// TIA Portal V16 export
// export: Created 2021-06-17T11:14:34.052257Z, ExportSetting WithDefaults, DisplayName Totally Integrated Automation Portal, DisplayVersion V16 Update 4, DisplayName TIA Portal Version Control Interface, DisplayVersion V16 Update 2, DisplayName TIA Portal Openness, DisplayVersion V16 Update 4, DisplayName SINAMICS Startdrive Advanced, DisplayVersion V16 Update 5, DisplayName SINAMICS Startdrive G130, G150, S120, S150, SINAMICS MV, S210, DisplayVersion V16 Update 5, DisplayName SINAMICS Startdrive G110M, G120, G120C, G120D, G120P, G115D, DisplayVersion V16 Update 5, DisplayName STEP 7 Professional, DisplayVersion V16 Update 4, DisplayName SIMATIC Energy Suite, DisplayVersion V16 Update 4, DisplayName STEP 7 Safety, DisplayVersion V16, DisplayName WinCC Advanced / Unified PC, DisplayVersion V16 Update 4, DisplayName SIMATIC Visualization Architect, DisplayVersion V16 Update 1
TYPE "UDT_ACB_ETI"
// stored: IsFailsafeCompliant false
   STRUCT
      ID : Int;   // MOT(ID=5001...6000)
      CLSID : Word := WORD#16#2110;   // Type of element
      Mode { ExternalAccessible := 'False'; ExternalVisible := 'False'; ExternalWritable := 'False'} : "Mode";
      State { ExternalAccessible := 'False'; ExternalVisible := 'False'; ExternalWritable := 'False'} : Struct   // Main state
         Error { ExternalAccessible := 'False'; ExternalVisible := 'False'; ExternalWritable := 'False'} : Bool;   // 1 = [1-level alarm] General alarm - Overall error
         Warning { ExternalAccessible := 'False'; ExternalVisible := 'False'; ExternalWritable := 'False'} : Bool;   // 1 = [2-level alarm] Warning
         Maintenance { ExternalAccessible := 'False'; ExternalVisible := 'False'; ExternalWritable := 'False'} : Bool;   // 1 = [3-level ] Maintenance
         Interlocked { ExternalAccessible := 'False'; ExternalVisible := 'False'; ExternalWritable := 'False'} : Bool;   // 1 = [Interlock] -Status interlock - Motor interlocked
         Ready { ExternalAccessible := 'False'; ExternalVisible := 'False'; ExternalWritable := 'False'} : Bool;   // 1 = Ready
         Closed { ExternalAccessible := 'False'; ExternalVisible := 'False'; ExternalWritable := 'False'} : Bool;   // 1 = Closed = IB_114_FeedbackClose+ QB_CmdCloseACB
         Opened { ExternalAccessible := 'False'; ExternalVisible := 'False'; ExternalWritable := 'False'} : Bool;   // 1 = Opened = IB_114_FeedbackOpen+ QB_CmdOpenACB
         Closing { ExternalAccessible := 'False'; ExternalVisible := 'False'; ExternalWritable := 'False'} : Bool;   // 1 = Closing - закривається
         Opening { ExternalAccessible := 'False'; ExternalVisible := 'False'; ExternalWritable := 'False'} : Bool;   // 1 = Opening - відкривається
         InCmdAutoClose { ExternalAccessible := 'False'; ExternalVisible := 'False'; ExternalWritable := 'False'} : Bool;   // 1 = Auto COMMAND - ACB to CLOSE
         InCmdAutoOpen { ExternalAccessible := 'False'; ExternalVisible := 'False'; ExternalWritable := 'False'} : Bool;   // 1 = Auto COMMAND - ACB to OPEN
         SigOutOpen { ExternalAccessible := 'False'; ExternalVisible := 'False'; ExternalWritable := 'False'} : Bool;   // StateTransferredTo physical output.Activate the output - QB_CmdCloseACB
         SigOutClose { ExternalAccessible := 'False'; ExternalVisible := 'False'; ExternalWritable := 'False'} : Bool;   // State transferred to physical output.Activate the output - QB_CmdOpenACB
      END_STRUCT;
      Alarm { ExternalAccessible := 'False'; ExternalVisible := 'False'; ExternalWritable := 'False'} : Struct
         InterlockingBypassed { ExternalAccessible := 'False'; ExternalVisible := 'False'; ExternalWritable := 'False'} : Bool;
         InterlockBypassed { ExternalAccessible := 'False'; ExternalVisible := 'False'; ExternalWritable := 'False'} : Bool;
         ErrTimeOut { ExternalAccessible := 'False'; ExternalVisible := 'False'; ExternalWritable := 'False'} : Bool;   // 1 = TimeOut
         ExtWarning { ExternalAccessible := 'False'; ExternalVisible := 'False'; ExternalWritable := 'False'} : Bool;   // 1 = External warning active + Warning
         ExtError { ExternalAccessible := 'False'; ExternalVisible := 'False'; ExternalWritable := 'False'} : Bool;   // 1 = External Fault is active + Error
         PreAlarm { ExternalAccessible := 'False'; ExternalVisible := 'False'; ExternalWritable := 'False'} : Bool;
         SystemFault { ExternalAccessible := 'False'; ExternalVisible := 'False'; ExternalWritable := 'False'} : Bool;   // 2^9 1 = Emergency SAFETY Motor Local switch OFF(Local disconnect OFF) +Error
         TripLT { ExternalAccessible := 'False'; ExternalVisible := 'False'; ExternalWritable := 'False'} : Bool;   // 2^10 0 = Motor Protector OK / 1 = Motor ProtectorTripped + Error
         TripST { ExternalAccessible := 'False'; ExternalVisible := 'False'; ExternalWritable := 'False'} : Bool;   // 2^11 0 = Clutch OK /1 = Clutch tripped + Error
         ErrClosing { ExternalAccessible := 'False'; ExternalVisible := 'False'; ExternalWritable := 'False'} : Bool;   // 2^12 1 = ÐŸÐ¾Ð¼Ð¸Ð»ÐºÐ° Ð·Ð°Ð¿ÑƒÑÐºÑƒ/ No signal from forward contactor + Error
         ErrOpening { ExternalAccessible := 'False'; ExternalVisible := 'False'; ExternalWritable := 'False'} : Bool;   // 2^141 = ÐŸÐ¾Ð¼Ð¸Ð»ÐºÐ° Ð·ÑƒÐ¿Ð¸Ð½ÐºÐ¸ / Motor doesn't stop / Switching time exceeded. + Error
         ErrPlaus { ExternalAccessible := 'False'; ExternalVisible := 'False'; ExternalWritable := 'False'} : Bool;   // 2^15 1=errorPlaus-Activation not plausible(switched on or switched off at the s
         MaintACT { ExternalAccessible := 'False'; ExternalVisible := 'False'; ExternalWritable := 'False'} : Bool;   // 2^6 1=Ðœaintenance-Limit Number object switching operations Reached + Maintenanc
         MaintTIME { ExternalAccessible := 'False'; ExternalVisible := 'False'; ExternalWritable := 'False'} : Bool;   // 2^7 1 = Ðœaintenance-Limit Operating time Reached + Maintenance
         EstopLocal { ExternalAccessible := 'False'; ExternalVisible := 'False'; ExternalWritable := 'False'} : Bool;   // 2^0 1 = Estop active + Error
         EstopHMI { ExternalAccessible := 'False'; ExternalVisible := 'False'; ExternalWritable := 'False'} : Bool;   // 2^0 1 = Estop active + Error
         FaultSuppyBox { ExternalAccessible := 'False'; ExternalVisible := 'False'; ExternalWritable := 'False'} : Bool;
      END_STRUCT;
      CMD : Int;   // 16#0100/16#0101/16#0102/16#0200/16#0201/16#0202/16#0300/16#0301/16#0302
      PRM : Struct
         W { ExternalAccessible := 'False'; ExternalVisible := 'False'; ExternalWritable := 'False'} : Struct
            ManLocalPirority { ExternalAccessible := 'False'; ExternalVisible := 'False'; ExternalWritable := 'False'; S7_SetPoint := 'True'} : Bool;   // 1 = HIGHT - enable from FC input/0 = LOW - enable from HMI
            AutoAskErrors { ExternalAccessible := 'False'; ExternalVisible := 'False'; ExternalWritable := 'False'; S7_SetPoint := 'True'} : Bool;   // 1 = Ð°Ð²Ñ‚Ð¾Ð¼Ð°Ñ‚Ð¸Ñ‡Ð½Ðµ Ð¿Ñ–Ð´Ñ‚Ð²ÐµÑ€Ð´Ð¶ÐµÐ½Ð½Ñ Ñ‚Ñ€Ð¸Ð²Ð¾Ð³
            LockExtModeChange { ExternalAccessible := 'False'; ExternalVisible := 'False'; ExternalWritable := 'False'; S7_SetPoint := 'True'} : Bool;
            InterlockBypass { ExternalAccessible := 'False'; ExternalVisible := 'False'; ExternalWritable := 'False'; S7_SetPoint := 'True'} : Bool;   // Interlocking obj bypassed / disable
            InterlockAutoReset { ExternalAccessible := 'False'; ExternalVisible := 'False'; ExternalWritable := 'False'; S7_SetPoint := 'True'} : Bool;
         END_STRUCT;
         enableExternalErrors { ExternalAccessible := 'False'; ExternalVisible := 'False'; ExternalWritable := 'False'; S7_SetPoint := 'True'} : Word := 16#FFFF;   // bit - 1 = enable
         bypassInterlocks { ExternalAccessible := 'False'; ExternalVisible := 'False'; ExternalWritable := 'False'; S7_SetPoint := 'True'} : Word := 16#FFFF;   // bit - 0 = Interlock Bypassed
         spTimeOut { S7_SetPoint := 'True'} : Int := 50;   // Monitoring time for ERROR ErrRunFRD ErrRunRVS ErrStop ErrPlaus (0.1sec)
         spTimeOnDelAuto { S7_SetPoint := 'True'} : Int := 50;   // Setpoint delay on time after start auto command (0.1sec)
         spTimeOffDelAuto { S7_SetPoint := 'True'} : Int := 50;   // Setpoint delay off time after stop auto command (0.1sec)
         spTimeRestart { S7_SetPoint := 'True'} : Int := 50;   // Час блокування повторного запуску (0.1sec)
         spTimeFixError { S7_SetPoint := 'True'} : Int := 50;   // Чac блокування скидання помилок дляїх фіксації в HMI (0.1sec.)
         spTimeCmdCloseOpen { S7_SetPoint := 'True'} : Int := 50;
         spMaintTimeOperPeriod { S7_SetPoint := 'True'} : DInt;   // Maintenance period - Operating time in hours 0=OFF (hour)
         spMaintActivPeriod { S7_SetPoint := 'True'} : DInt;   // Maintenance period-number object activated switches/switching operations 0=OFF
         spare48 { S7_SetPoint := 'True'} : Int;
      END_STRUCT;
      Counters { ExternalWritable := 'False'} : Struct   // Лічильники
         cvMaintTimeOperPeriodTOT { ExternalWritable := 'False'; S7_SetPoint := 'True'} : DInt;   // Total Time Operating time in hours
         cvMaintTimeOperPeriodrLAST { ExternalWritable := 'False'; S7_SetPoint := 'True'} : DInt;   // Operating time in hours from last maintenance
         cvMaintActivPeriodTOT { ExternalWritable := 'False'; S7_SetPoint := 'True'} : DInt;   // Ð¢otal counter object activated switches/switching operations
         cvMaintActivPeriodLAST { ExternalWritable := 'False'; S7_SetPoint := 'True'} : DInt;   // Counter object activated switches/switching operations from last maintenance
         cvError { ExternalWritable := 'False'; S7_SetPoint := 'True'} : DInt;   // Лічильник кількості помилок
         cvWarning { ExternalWritable := 'False'; S7_SetPoint := 'True'} : DInt;   // Лічильник кількості полпереджень
      END_STRUCT;
      Simualtion { ExternalAccessible := 'False'; ExternalVisible := 'False'; ExternalWritable := 'False'} : Struct
         Enable { ExternalAccessible := 'False'; ExternalVisible := 'False'; ExternalWritable := 'False'} : Struct
            IB_EstopLocal { ExternalAccessible := 'False'; ExternalVisible := 'False'; ExternalWritable := 'False'} : Bool;
            IB_EstopHMI { ExternalAccessible := 'False'; ExternalVisible := 'False'; ExternalWritable := 'False'} : Bool;
            IB_SuppyBox_Ok { ExternalAccessible := 'False'; ExternalVisible := 'False'; ExternalWritable := 'False'} : Bool;
            IB_15_TripLT { ExternalAccessible := 'False'; ExternalVisible := 'False'; ExternalWritable := 'False'} : Bool;
            IB_26_SystemAlarm { ExternalAccessible := 'False'; ExternalVisible := 'False'; ExternalWritable := 'False'} : Bool;
            IB_25_TripST { ExternalAccessible := 'False'; ExternalVisible := 'False'; ExternalWritable := 'False'} : Bool;
            IB_06_PreAlarmPTA { ExternalAccessible := 'False'; ExternalVisible := 'False'; ExternalWritable := 'False'} : Bool;
            IW_Interlocks { ExternalAccessible := 'False'; ExternalVisible := 'False'; ExternalWritable := 'False'} : Bool;
            IW_ExternalError { ExternalAccessible := 'False'; ExternalVisible := 'False'; ExternalWritable := 'False'} : Bool;
            IB_ExternalWarning { ExternalAccessible := 'False'; ExternalVisible := 'False'; ExternalWritable := 'False'} : Bool;
            IB_CmdAutoClose { ExternalAccessible := 'False'; ExternalVisible := 'False'; ExternalWritable := 'False'} : Bool;
            IB_CmdAutoOpen { ExternalAccessible := 'False'; ExternalVisible := 'False'; ExternalWritable := 'False'} : Bool;
            IB_CmdManualLocal { ExternalAccessible := 'False'; ExternalVisible := 'False'; ExternalWritable := 'False'} : Bool;
            IB_CmdManLocalClose { ExternalAccessible := 'False'; ExternalVisible := 'False'; ExternalWritable := 'False'} : Bool;
            IB_CmdManLocalOpen { ExternalAccessible := 'False'; ExternalVisible := 'False'; ExternalWritable := 'False'} : Bool;
         END_STRUCT;
         spTimeSimFeedbackOnDelay { ExternalAccessible := 'False'; ExternalVisible := 'False'; ExternalWritable := 'False'; S7_SetPoint := 'True'} : Int := 20;
      END_STRUCT;
      HMI_DATA { ExternalWritable := 'False'} : "ACB_ETI_HMI";
   END_STRUCT;
END_TYPE
